(*
SPDX-FileCopyrightText: © 2026 Oleksandr Tiutyk <trofimich@gmail.com>
SPDX-License-Identifier: MIT
License: https://opensource.org/license/mit
*)

(*!
<summary>
Defines the root automation controller capable of coordinating child components and controller plugins.
</summary>
<description>Indexed Try lookups return borrowed interfaces or null and do not propagate exceptions.</description>
*)

INTERFACE IAutomationController EXTENDS IParentAutomationComponent

{attribute 'monitoring' := 'call'}
PROPERTY FINAL PluginCount : TOF_Core.INT_LENGTH
GET
END_GET
END_PROPERTY

(*!
<summary>Returns a borrowed plugin by its zero-based index.</summary>
<description>
Returns null when the entry is unavailable, the index is out of range or a nested call raises an exception.
Fatal allocation observations return null and leave the fatal latch set for the outer task boundary.
Does not transfer ownership or extend lifetime. Implementations must not propagate exceptions.
</description>
*)
METHOD TryGetPluginByIndex : IAutomationControllerPlugin
VAR_INPUT
	index : TOF_Core.INT_INDEX;
END_VAR
END_METHOD

END_INTERFACE

(* stored: Version 1.1.0.1
   Itf IAutomationController: Id {0b4e8e80-e173-49c5-86a2-54e893b4c200}
   Property PluginCount: Id {b6aa27af-1d06-4aea-8e2c-3eda3657bf33}
   Get Get: Id {a7f23203-43c8-446f-82f0-3a72173748c8}
   Method TryGetPluginByIndex: Id {ba60eef3-9279-4fda-8f5e-7bace35abbbc} *)
